PROGRAM GL2_Transfer
VAR
	
	
	GL1_RD: SRoll_Door;
	GL2_PASSSED_ROLL_DOOR : BOOL;
	RUN_FWD_TO_GL6_BIT : BOOL; // GL2 OCCUPIED, GL6 REQUESTING PART, RUN TO GL6 POSITION
	RUN_FWD_TO_GL8_BIT : BOOL; // GL2 OCCUPIED, GL8 REQUESTING PART, RUN TO GL8 POSITION
	RUN_REV_TO_GL5_BIT : BOOL; //GL2 EMPTY, GL2 REQUESTING PART, RUN TO GL5 POSITION
	TOF_occupied_delay_off: tof;
	TOF_occupied_delay_of_elapsed: TIME;
	
END_VAR
VAR // added by the converter: edge detectors and wires of the graphical bodies
    _w1 : BOOL;
END_VAR

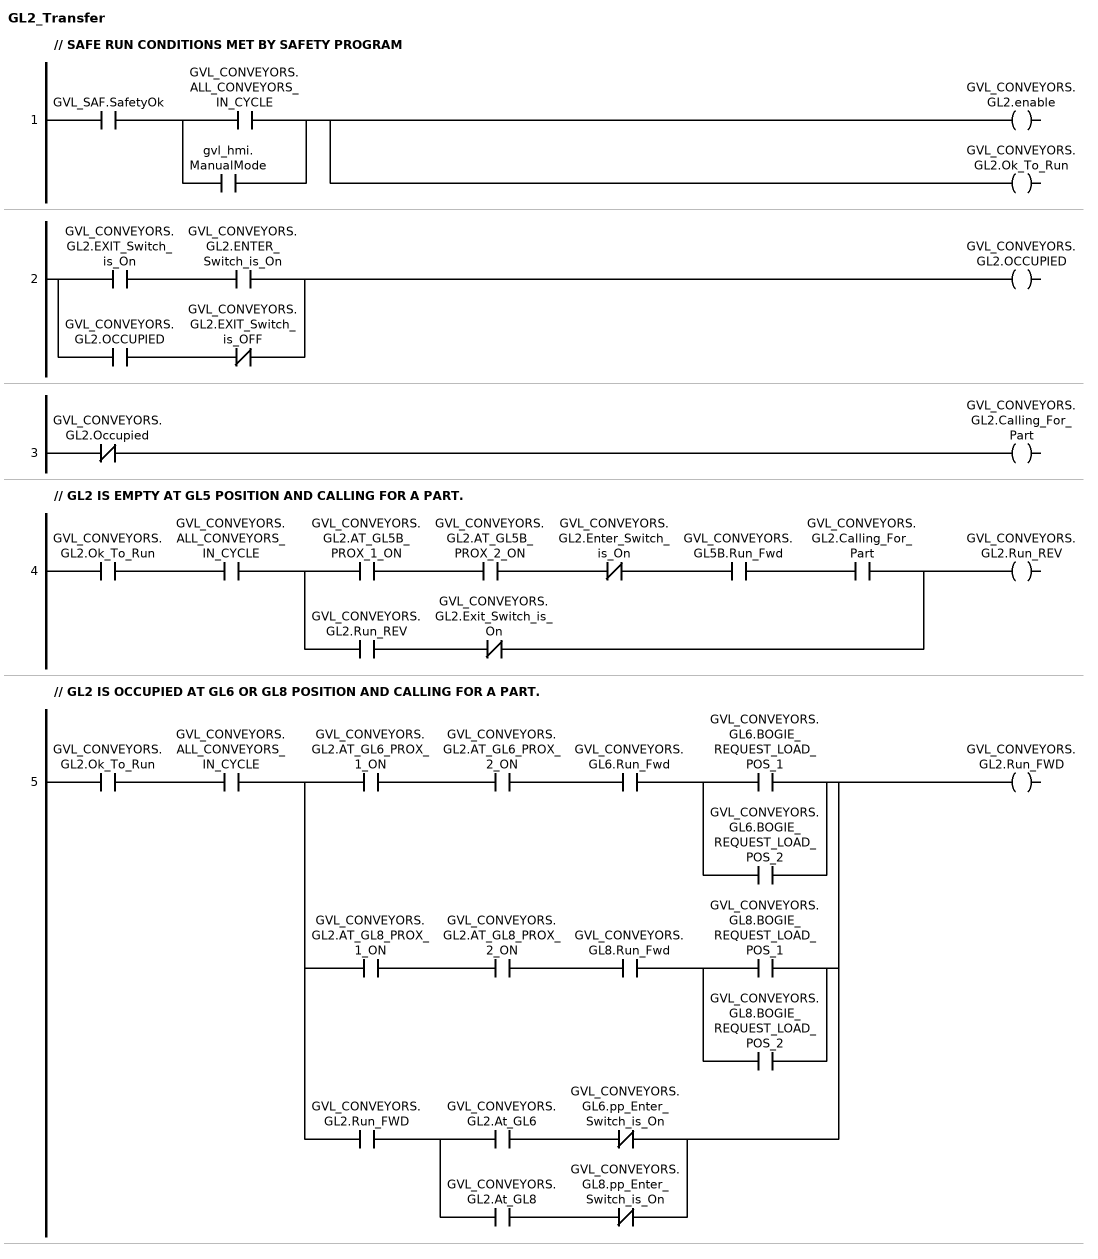
// NETWORK 1: // SAFE RUN CONDITIONS MET BY SAFETY PROGRAM
_w1 := GVL_SAF.SafetyOk AND (GVL_CONVEYORS.ALL_CONVEYORS_IN_CYCLE OR gvl_hmi.ManualMode);
GVL_CONVEYORS.GL2.enable := _w1;
GVL_CONVEYORS.GL2.Ok_To_Run := _w1;

// NETWORK 2
GVL_CONVEYORS.GL2.OCCUPIED := GVL_CONVEYORS.GL2.EXIT_Switch_is_On AND GVL_CONVEYORS.GL2.ENTER_Switch_is_On OR GVL_CONVEYORS.GL2.OCCUPIED AND NOT GVL_CONVEYORS.GL2.EXIT_Switch_is_OFF;

// NETWORK 3
GVL_CONVEYORS.GL2.Calling_For_Part := NOT GVL_CONVEYORS.GL2.Occupied;

// NETWORK 4: // GL2 IS EMPTY AT GL5 POSITION AND CALLING FOR A PART.
GVL_CONVEYORS.GL2.Run_REV := GVL_CONVEYORS.GL2.Ok_To_Run AND GVL_CONVEYORS.ALL_CONVEYORS_IN_CYCLE AND (GVL_CONVEYORS.GL2.AT_GL5B_PROX_1_ON AND GVL_CONVEYORS.GL2.AT_GL5B_PROX_2_ON AND NOT GVL_CONVEYORS.GL2.Enter_Switch_is_On AND GVL_CONVEYORS.GL5B.Run_Fwd AND GVL_CONVEYORS.GL2.Calling_For_Part OR GVL_CONVEYORS.GL2.Run_REV AND NOT GVL_CONVEYORS.GL2.Exit_Switch_is_On);

// NETWORK 5: // GL2 IS OCCUPIED AT GL6 OR GL8 POSITION AND CALLING FOR A PART.
GVL_CONVEYORS.GL2.Run_FWD := GVL_CONVEYORS.GL2.Ok_To_Run AND GVL_CONVEYORS.ALL_CONVEYORS_IN_CYCLE AND (GVL_CONVEYORS.GL2.AT_GL6_PROX_1_ON AND GVL_CONVEYORS.GL2.AT_GL6_PROX_2_ON AND GVL_CONVEYORS.GL6.Run_Fwd AND (GVL_CONVEYORS.GL6.BOGIE_REQUEST_LOAD_POS_1 OR GVL_CONVEYORS.GL6.BOGIE_REQUEST_LOAD_POS_2) OR GVL_CONVEYORS.GL2.AT_GL8_PROX_1_ON AND GVL_CONVEYORS.GL2.AT_GL8_PROX_2_ON AND GVL_CONVEYORS.GL8.Run_Fwd AND (GVL_CONVEYORS.GL8.BOGIE_REQUEST_LOAD_POS_1 OR GVL_CONVEYORS.GL8.BOGIE_REQUEST_LOAD_POS_2) OR GVL_CONVEYORS.GL2.Run_FWD AND (GVL_CONVEYORS.GL2.At_GL6 AND NOT GVL_CONVEYORS.GL6.pp_Enter_Switch_is_On OR GVL_CONVEYORS.GL2.At_GL8 AND NOT GVL_CONVEYORS.GL8.pp_Enter_Switch_is_On));

END_PROGRAM

(* stored: Version 1.1.0.1, ProductVersion 3.1.4024.12
   POU GL2_Transfer: Id {00c5fb8a-74fe-43e1-b6a4-7d53354e0e95}, SpecialFunc None *)
